// Represents the year as a four-digit value (e.g., 2024).
TYPE T_Year : UINT; END_TYPE

(* stored: Version 1.1.0.1
   DUT T_Year: Id {4c85ceef-45f0-076c-2555-da3b6a070ea4} *)
